ABB RobotStudio station: sesion6_EstacionDePartidaclase.rspag

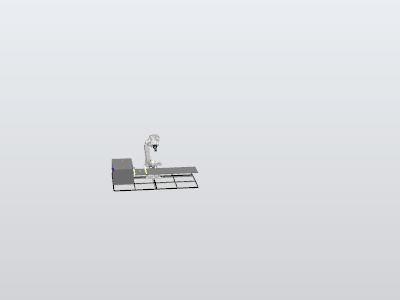
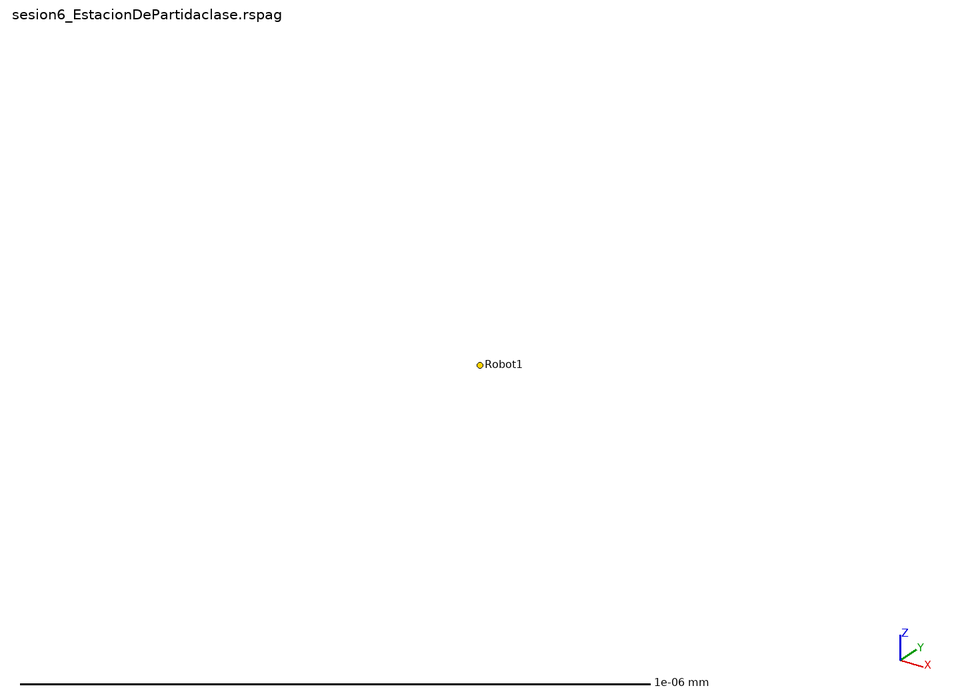
[picture v1: parts stored in the station drawn from their meshes, with robot base, taught points and paths (robot models come from the ABB library and are not in the file)]
--- station ---
Station sesion7_EstacionDePartida_1 (saved by RobotStudio 24.1.10713.1)
Controller Sistema6
  mechanical unit ROB_1: Robot1, 6 joints, base frame (0, 0, 0) mm
Layout (positions relative to the parent item):
  - Ventosa [mechanism] at (1635.7, 0, 1955) mm, rotated rx 180 ry 60 rz 180 deg
      TCP Ventosa at (0, 0, 200) mm
      links: PiezaVentosa
  - Robot1 [mechanism, from %ABB.RobotStudio.Models.IRB6640%\IRB6640_180_255_G_04.rslib] at (0, 0, 0) mm; joint values [0, 0, 0, 0, 0.5236, 0] (rad or m)
  - CI_VentosaVacuostato [smart component]
      signals: DI ActivaVentosa, DO Vacuostato
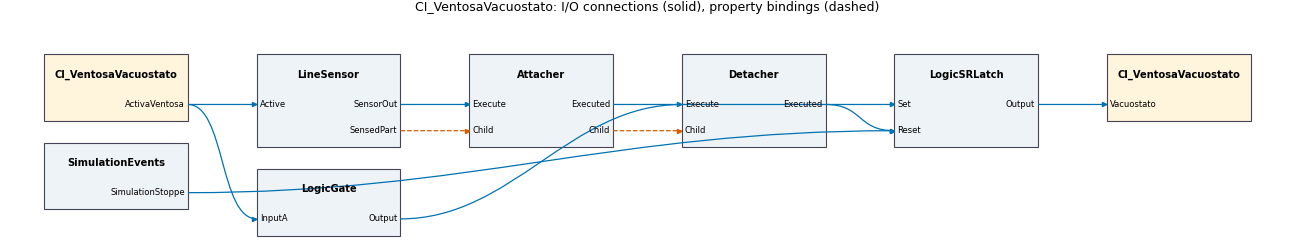
      connections:
        CI_VentosaVacuostato.ActivaVentosa -> LineSensor.Active
        LineSensor.SensorOut -> Attacher.Execute
        Attacher.Executed -> LogicSRLatch.Set
        LogicSRLatch.Output -> CI_VentosaVacuostato.Vacuostato
        Detacher.Executed -> LogicSRLatch.Reset
        SimulationEvents.SimulationStopped -> LogicSRLatch.Reset
        CI_VentosaVacuostato.ActivaVentosa -> LogicGate.InputA
        LogicGate.Output -> Detacher.Execute
        LineSensor.SensedPart => Attacher.Child
        Attacher.Child => Detacher.Child
    - LineSensor [smart component, from Components\LineSensor.rslib] at (1808.91, 0, 1855) mm, rotated rx 180 ry 60 rz 180 deg
        properties: Start=[0 0 -0.002]; End=[0 0 0.02]; Radius=0.002; SensedPart=(none); SensedPoint=[1.50000012207031 0.500000030517578 0.85]; Length=0.022; Tag=(none)
      - _sensorPart_ [part], size 4 x 4 x 22 mm
    - SimulationEvents [smart component, from Components\SimulationEvents.rslib]
    - LogicSRLatch [smart component, from Components\LogicSRLatch.rslib]
    - Attacher [smart component, from Components\Attacher.rslib]
        properties: Parent=Ventosa; Flange=0; Child=(none); Mount=false; Offset=[0 0 0]; Orientation=[0 0 0]
    - Detacher [smart component, from Components\Detacher.rslib]
        properties: Child=(none); KeepPosition=true
    - LogicGate [smart component, from Components\LogicGate.rslib]
        properties: Operator=NOT; Delay=0.1
  - MesaPaletizadoParteIzq [part], size 1000 x 1000 x 750 mm
  - MesaPaletizadoParteDer [part], size 1000 x 1000 x 750 mm
  - cintaTransportadora [part], size 1000 x 3000 x 30 mm
  - PiezaLarga [part], size 500 x 1000 x 30 mm
  - PiezaCorta [part], size 500 x 500 x 30 mm
  - CI_SensoresCinta [smart component]
      signals: DI ActivaSensores, DO FinalCintaDetectado, DO PiezaLargaDetectada
      connections:
        CI_SensoresCinta.ActivaSensores -> LineSensorFinalCinta.Active
        CI_SensoresCinta.ActivaSensores -> LineSensorPiezaLarga.Active
        LineSensorPiezaLarga.SensorOut -> CI_SensoresCinta.PiezaLargaDetectada
        LineSensorFinalCinta.SensorOut -> CI_SensoresCinta.FinalCintaDetectado
    - LineSensorFinalCinta [smart component, from Components\LineSensor.rslib]
        properties: Start=[1 -1 0.765]; End=[2 -1 0.765]; Length=1; Radius=0.002; Tag=(none); SensedPart=(none); SensedPoint=[0 0 0]
      - _sensorPart_ [part], size 1000 x 4 x 4 mm
    - LineSensorPiezaLarga [smart component, from Components\LineSensor.rslib]
        properties: Start=[1 -0.45 0.765]; End=[2 -0.45 0.765]; Length=1; Radius=0.002; Tag=(none); SensedPart=(none); SensedPoint=[0 0 0]
      - _sensorPart_ [part], size 1000 x 4 x 4 mm
  - CI_CintaTransportadora [smart component]
      signals: DI PideNuevaPieza, DI MueveCinta, DI Desencolar
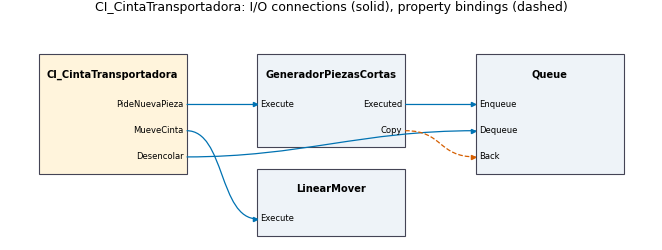
      connections:
        GeneradorPiezasCortas.Executed -> Queue.Enqueue
        CI_CintaTransportadora.PideNuevaPieza -> GeneradorPiezasCortas.Execute
        CI_CintaTransportadora.MueveCinta -> LinearMover.Execute
        CI_CintaTransportadora.Desencolar -> Queue.Dequeue
        GeneradorPiezasCortas.Copy => Queue.Back
    - GeneradorPiezasCortas [smart component, from Components\Source.rslib]
        properties: Source=PiezaCorta; Copy=(none); Parent=(none); Position=[1.25 1.5 0.75]; Orientation=[0 0 0]; Transient=false; PhysicsBehavior=-1
    - LinearMover [smart component, from Components\LinearMover.rslib]
        properties: Object=Queue; Direction=[0 -0.001 0]; Speed=0.2; Reference=Global; ReferenceObject=(none)
    - Queue [smart component, from Components\Queue.rslib]
        properties: Back=(none); Front=(none); Queue=; NumberOfObjects=0
Attachment: Ventosa is attached to Robot1 / Link6
Attachment: LineSensor is attached to Ventosa / PiezaVentosa
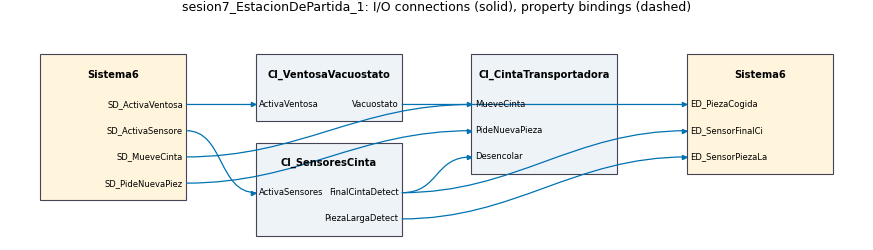
Station logic (signal -> signal, property => property):
  CI_VentosaVacuostato.Vacuostato -> Sistema6.ED_PiezaCogida
  Sistema6.SD_ActivaVentosa -> CI_VentosaVacuostato.ActivaVentosa
  CI_SensoresCinta.FinalCintaDetectado -> Sistema6.ED_SensorFinalCinta
  CI_SensoresCinta.PiezaLargaDetectada -> Sistema6.ED_SensorPiezaLarga
  Sistema6.SD_ActivaSensores -> CI_SensoresCinta.ActivaSensores
  Sistema6.SD_MueveCinta -> CI_CintaTransportadora.MueveCinta
  Sistema6.SD_PideNuevaPieza -> CI_CintaTransportadora.PideNuevaPieza
  CI_SensoresCinta.FinalCintaDetectado -> CI_CintaTransportadora.Desencolar
Targets, tools, work objects and paths stored in the station and not in the controller backup, written as RAPID:
! task T_ROB1
MODULE CalibData
  TASK PERS wobjdata WO_Paletizado:=[FALSE,TRUE,"",[[1000,-2000,750],[0.707106781,0,0,0.707106781]],[[0,0,0],[1,0,0,0]]];
  TASK PERS wobjdata WO_CintaTransportadora:=[FALSE,TRUE,"",[[1000,-1000,750],[1,0,0,0]],[[0,0,0],[1,0,0,0]]];
ENDMODULE

! task T_ROB1
MODULE Module1
  CONST robtarget pReposo:=[[1808.910161514,0,1855],[0.5,0,0.866025404,0],[0,0,0,0],[9E+09,9E+09,9E+09,9E+09,9E+09,9E+09]];
  CONST robtarget pBasePalePiezasCortas:=[[500,500,0],[0,1,0,0],[0,0,0,0],[9E+09,9E+09,9E+09,9E+09,9E+09,9E+09]];
  CONST robtarget pBasePalePiezasLargas:=[[500,1500,0],[0,1,0,0],[0,0,0,0],[9E+09,9E+09,9E+09,9E+09,9E+09,9E+09]];
  CONST robtarget pBaseCogidaPiezaLarga:=[[500,500,0],[0,0,1,0],[0,0,0,0],[9E+09,9E+09,9E+09,9E+09,9E+09,9E+09]];
  CONST robtarget pBaseCogidaPiezaCorta:=[[500,250,0],[0,0,1,0],[0,0,0,0],[9E+09,9E+09,9E+09,9E+09,9E+09,9E+09]];
ENDMODULE


--- Backups/Sistema6/RAPID/TASK1/PROGMOD/CalibData.mod ---
MODULE CalibData
	PERS tooldata Ventosa:=[TRUE,[[0,0,200],[1,0,0,0]],[1,[0,0,125],[1,0,0,0],0.002,0.002,0.0013]];
ENDMODULE

--- Backups/Sistema6/RAPID/TASK1/PROGMOD/Module1.mod ---
MODULE Module1
ENDMODULE

--- Backups/Sistema6/RAPID/TASK1/SYSMOD/LINKEDM.sys ---
%%%
  VERSION:1
  LANGUAGE:ENGLISH
%%%

MODULE LINKEDM (SYSMODULE)

! FOLLOWER
!     Name of electronically linked follower axis used by operator at teach pendent.
      PERS string l_f_axis_name{5}       :=  ["",  "", "", "", ""];

!     Name of the mechanical unit for follower axis.
      PERS string l_f_mecunt_n{5}  :=  ["", "", "", "", ""];

!     Linked follower axis number in the mechanical unit (first axis in mech. unit is number 1).
      PERS num l_f_axis_no{5}      :=  [0,          0,   0,  0,  0];

! MASTER
!     Name of the mechanical unit for linked master axis.
      PERS string l_m_mecunt_n{5} :=  ["", "", "", "", ""];

!     Linked master axis number in the mechanical unit (first axis in mech. unit is number 1).
!     See axis number table in documentation for different master mechanical units.
      PERS num l_m_axis_no{5}     :=  [0,  0,  0,  0,  0];

! POSITION OFFSET
!     The increase of the allowed offset position between the master and follower
!     positions, used when starting AUTO mode. As soon as the offset is decreased
!     the old configurated parameter is used.
!     Example: 3 => the configurated value of allowed offset is increased 3 times.
      PERS num offset_ratio{5}       :=  [10,  10,   10,  10,  10];

! SPEED RATIO
!     Speed_ratio used in AUTO and JOG modes [ very_slow   slow    normal    fast]
!     Value 1 = max allowed manual speed.
      CONST num speed_ratio {20}      := [0.01, 0.01, 0.01, 0.01, 0.01,
                                          0.05, 0.05, 0.05, 0.05, 0.05,
                                          0.20, 0.20, 0.20, 0.20, 0.20,
                                          1.00, 1.00, 1.00, 1.00, 1.00];

! STEP SIZE
!     Displacement position used in JOG mode for each activation of positive or
!     negative movement.                  [very_short    short   normal   long]
!     Unit degees or meter.
      CONST num displacement {20}     := [0.001, 0.001, 0.001, 0.001, 0.001,
                                          0.005, 0.005, 0.005, 0.005, 0.005,
                                          0.020, 0.020, 0.020, 0.020, 0.020,
                                          0.100, 0.100, 0.100, 0.100, 0.100];


!-------------------------------------------------------------
 PROC Linked_m ()
      Linked_m_exe ;
 ENDPROC
ENDMODULE

--- Backups/Sistema6/SYSPAR/EIO.cfg ---
EIO:CFG_1.0:6:1::
#
INDUSTRIAL_NETWORK:

      -Name "DeviceNet" -Label "DeviceNet Master/Slave Network" -Address "2"
#
DEVICENET_DEVICE:

      -Name "MiDeviceNet" -Label "MiDeviceNet"
#
DEVICENET_INTERNAL_DEVICE:

      -Name "DN_Internal_Device" -VendorName "ABB Robotics"\
      -ProductName "DeviceNet Internal Slave Device"
#
EIO_SIGNAL:

      -Name "ED_PiezaCogida" -SignalType "DI" -Device "MiDeviceNet"\
      -Label "ED_PiezaCogida" -DeviceMap "0" -Access "All"

      -Name "SD_ActivaVentosa" -SignalType "DO" -Device "MiDeviceNet"\
      -Label "SD_ActivaVentosa" -DeviceMap "0" -Access "All"

      -Name "ED_SensorFinalCinta" -SignalType "DI" -Device "MiDeviceNet"\
      -Label "ED_SensorFinalCinta" -DeviceMap "1" -Access "All"

      -Name "ED_SensorPiezaLarga" -SignalType "DI" -Device "MiDeviceNet"\
      -Label "ED_SensorPiezaLarga" -DeviceMap "2" -Access "All"

      -Name "SD_ActivaSensores" -SignalType "DO" -Device "MiDeviceNet"\
      -Label "SD_ActivaSensores" -DeviceMap "1" -Access "All"

      -Name "SD_MueveCinta" -SignalType "DO" -Device "MiDeviceNet"\
      -Label "SD_MueveCinta" -DeviceMap "2" -Access "All"

      -Name "SD_PideNuevaPieza" -SignalType "DO" -Device "MiDeviceNet"\
      -Label "SD_PideNuevaPieza" -DeviceMap "3" -Access "All"
